// TwinCAT 3 PLC project EventsHistoricalSimple
// ProgramVersion: 3.1.4020.4
// CompilerDefines: VISU_USEWSTRING
// libraries:
//   Tc2_Standard, * (Beckhoff Automation GmbH)
//   Tc2_System, * (Beckhoff Automation GmbH)
//   Tc2_Utilities, * (Beckhoff Automation GmbH)
//   Tc3_Module, * (Beckhoff Automation GmbH)
//   VisuDialogs, * (System)
// project tree:
//   DUTsEventsHS/ ST_EventDefinition.TcDUT, ST_EventHistoricalSimple.TcDUT, ST_EventHistoricalSimplePersistent.TcDUT
//   / GlobalTextList.TcGTLO, PlcTask.TcTTO, Visualization Manager.TcVMO (not stored), VISU_TASK.TcTTO
//   GVLsEventsHS/ GVL_EHS.TcGVL, GVL_EHSP.TcGVL
//   POUsEventsHS/POUsEventsHS/Functions/ F_RESET_Event.TcPOU, F_SET_Event.TcPOU
//   POUsEventsHS/POUsEventsHS/ P_EventsHS.TcPOU, P_EventsDefinitionHS.TcPOU, P_EventsHandlingHS.TcPOU, P_EventsVisuHS.TcPOU
//   POUsEventsHS/ MAIN.TcPOU
//   VISUsEventsHS/ VISU_EventsHistoricalSimple.TcVIS
// real-time tasks:
//   TASK PlcTask: cycle T#10ms, priority 20, ADS port 350
//   TASK VISU_TASK: cycle T#100000us, priority 30, ADS port 351

CONFIGURATION EventsHistoricalSimple
    RESOURCE PLC ON TwinCAT3
        TASK PlcTask(INTERVAL := T#10ms, PRIORITY := 20);
        TASK VISU_TASK(INTERVAL := T#100000us, PRIORITY := 30);
        PROGRAM MAIN WITH PlcTask : MAIN;
        PROGRAM VisuElems_Visu_Prg WITH VISU_TASK : VisuElems.Visu_Prg;
    END_RESOURCE
END_CONFIGURATION

// ---- DUTsEventsHS/ST_EventDefinition.TcDUT
//==================================================================================================
//							Beckhoff Automation Poland
//									23.05.2017
//	Struktura zawierajaca definicje zdarzenia
// 	v1.0	|| TC v 3.1.4020.32		|| - pierwsza wersja
//==================================================================================================
TYPE ST_EventDefinition :
STRUCT
	dwClass									: DWORD;
	dwParam									: DWORD;
	wsMessage								: WSTRING(80);
	bActive									: BOOL;
END_STRUCT
END_TYPE

// ---- DUTsEventsHS/ST_EventHistoricalSimple.TcDUT
//==================================================================================================
//							Beckhoff Automation Poland
//									23.05.2017
//	Struktura zawierajaca zdarzenie - pelne informacje, np. do wizualizacji
// 	v1.0	|| TC v 3.1.4020.32		|| - pierwsza wersja
//==================================================================================================
TYPE ST_EventHistoricalSimple :
STRUCT
	dwID									: DWORD;
	dwParam									: DWORD;
	dwClass									: DWORD;
	dtDateBegin								: DT;
	dtDateEnd								: DT;
	wsMessage								: WSTRING(80);
	dwColor									: UDINT;
END_STRUCT
END_TYPE

// ---- DUTsEventsHS/ST_EventHistoricalSimplePersistent.TcDUT
//==================================================================================================
//							Beckhoff Automation Poland
//									23.05.2017
//	Struktura zawierajaca zane do przechowania zdarzenia w pamieci
// 	v1.0	|| TC v 3.1.4020.32		|| - pierwsza wersja
//==================================================================================================
TYPE ST_EventHistoricalSimplePersistent :
STRUCT
	dwID									: DWORD;
	dwParam									: DWORD;
	dwClass									: DWORD;
	dtDateBegin								: DT;
	dtDateEnd								: DT;
END_STRUCT
END_TYPE

// ---- GVLsEventsHS/GVL_EHS.TcGVL
//==================================================================================================
//							Beckhoff Automation Poland
//									23.05.2017
// 	v1.0	|| TC v 3.1.4020.32		|| - pierwsza wersja
//==================================================================================================
{attribute 'qualified_only'}
VAR_GLOBAL CONSTANT
	diEventsDefinition						: DINT 	:= 50;				// Rozmiar tablicy definicji zdarzen, powinna byc w zakresie 5..1000
	diNoOfEvents							: DINT 	:= 100;				// Rozmiar tablicy zdarzen historycznych, powinna byc w zakresie 5..1000
END_VAR
VAR_GLOBAL
	stActTime								: TIMESTRUCT;				// Aktualny czas sytemowy w formie struktury
	dtActTime								: DT;						// Aktualny czas sytemowy
	arrEventDefinition 						: ARRAY [1..GVL_EHS.diEventsDefinition] OF ST_EventDefinition;
	arrEventVisu							: ARRAY [1..GVL_EHS.diNoOfEvents] OF ST_EventHistoricalSimple;		// Pokazywane na wizualizacji - po filtracji
	dwLanguageId							: DWORD := 1033;			// Kod jezyka wyswietlania - Microsoft Locale ID Values
END_VAR

// ---- GVLsEventsHS/GVL_EHSP.TcGVL
//==================================================================================================
//							Beckhoff Automation Poland
//									23.05.2017
// 	v1.0	|| TC v 3.1.4020.32		|| - pierwsza wersja
//==================================================================================================
{attribute 'qualified_only'}
VAR_GLOBAL PERSISTENT
	arrEvent								: ARRAY [1..GVL_EHS.diNoOfEvents] OF ST_EventHistoricalSimplePersistent;
END_VAR

// ---- POUsEventsHS/MAIN.TcPOU
PROGRAM MAIN
VAR
	tonWritePersistent						: TON;
	fbPersistent 							: FB_WritePersistentData;
END_VAR

tonWritePersistent(IN:= NOT tonWritePersistent.Q, PT:= T#1M, Q=> , ET=> );		// Zapis persistentow
fbPersistent(PORT:= 851, START:= tonWritePersistent.Q);							// Zapis persistentow
P_EventsHS();

END_PROGRAM

// ---- POUsEventsHS/POUsEventsHS/P_EventsHS.TcPOU
//==================================================================================================
//							Beckhoff Automation Poland
//									23.05.2017
//	Program obslugujacy proste alarmy historyczne.
//	W opcjach wizualizacji trzeba wybrac use uniceode strings i use current visu variable
// 	v1.0	|| TC v 3.1.4020.32		|| - pierwsza wersja
//==================================================================================================
PROGRAM P_EventsHS
VAR
	fbLocalSystemTime						: FB_LocalSystemTime;
	bEventTableSizeError					: BOOL;					// Niewlasciwy rozmiar tablicy zdarzen - sprawdz GVL_EHS.diNoOfEvents
	bEventDefinitionSizeError				: BOOL;					// Niewlasciwy rozmiar tablicy zdarzen - sprawdz GVL_EHS.diEventsDefinition
END_VAR

fbLocalSystemTime(bEnable:= TRUE, systemTime=> GVL_EHS.stActTime);
GVL_EHS.dtActTime 							:= SYSTEMTIME_TO_DT(GVL_EHS.stActTime);

P_EventsDefinitionHS ();

bEventDefinitionSizeError 					:= GVL_EHS.diEventsDefinition < 5 OR GVL_EHS.diEventsDefinition > 1000;
bEventTableSizeError 						:= GVL_EHS.diNoOfEvents < 5 OR GVL_EHS.diNoOfEvents > 1000;

IF NOT bEventDefinitionSizeError AND NOT bEventTableSizeError THEN
	IF fbLocalSystemTime.bValid THEN
		P_EventsHandlingHS();
	END_IF
	// Visu i filtry
	P_EventsVisuHS();	
END_IF

END_PROGRAM

// ---- POUsEventsHS/POUsEventsHS/P_EventsDefinitionHS.TcPOU
//==================================================================================================
//							Beckhoff Automation Poland
//									23.05.2017
//	Program definiujacy zdarzenia - musi byc dostosowany do aplikacji
//	W pierwszym cyklu definiowane sa klasy
//	Zmiana jezyka na zdarzenie i w pierwszym cyklu
//	Wykrywanie aktywnosci zdarzenia i parametru - cykliczne
// 	v1.0	|| TC v 3.1.4020.32		|| - pierwsza wersja
//==================================================================================================
PROGRAM P_EventsDefinitionHS
VAR
	bFirstCycle 							: BOOL := TRUE;
	dwPreviousLanguageID					: DWORD;
END_VAR

// Class
IF bFirstCycle THEN
	ACT_ClassDefinition();
	bFirstCycle 							:= FALSE;
END_IF

// Language
ACT_Language();

// Active
ACT_Active();

ACTION ACT_1033_US:
GVL_EHS.arrEventDefinition[1].wsMessage	 	:= "Alarm Message 1";
GVL_EHS.arrEventDefinition[2].wsMessage 	:= "Alarm Message 2";
GVL_EHS.arrEventDefinition[31].wsMessage 	:= "Warning Message 1";
GVL_EHS.arrEventDefinition[32].wsMessage 	:= "Warning Message 2";
GVL_EHS.arrEventDefinition[41].wsMessage 	:= "Message 1";
GVL_EHS.arrEventDefinition[42].wsMessage 	:= "Message 2";
END_ACTION

ACTION ACT_1045_PL:
GVL_EHS.arrEventDefinition[1].wsMessage		:= "Tekst alarmu 1";
GVL_EHS.arrEventDefinition[2].wsMessage		:= "śćąęźżółń 2";
GVL_EHS.arrEventDefinition[31].wsMessage	:= "Tekst ostrzeżenia 1";
GVL_EHS.arrEventDefinition[32].wsMessage	:= "Tekst ostrzeżenia 2";
GVL_EHS.arrEventDefinition[41].wsMessage	:= "Komunikat 1";
GVL_EHS.arrEventDefinition[42].wsMessage	:= "Komunikat 2";
END_ACTION

ACTION ACT_Active:
GVL_EHS.arrEventDefinition[1].bActive; // S=;
GVL_EHS.arrEventDefinition[1].bActive;// R=;
GVL_EHS.arrEventDefinition[1].dwParam := 1;
GVL_EHS.arrEventDefinition[2].bActive;
GVL_EHS.arrEventDefinition[2].dwParam := 2;
GVL_EHS.arrEventDefinition[31].bActive;
GVL_EHS.arrEventDefinition[31].dwParam := 3;
GVL_EHS.arrEventDefinition[32].bActive;
GVL_EHS.arrEventDefinition[32].dwParam := 4;
GVL_EHS.arrEventDefinition[41].bActive;
GVL_EHS.arrEventDefinition[41].dwParam := 5;
GVL_EHS.arrEventDefinition[42].bActive;
GVL_EHS.arrEventDefinition[42].dwParam;
END_ACTION

ACTION ACT_ClassDefinition:
// Error - 0
GVL_EHS.arrEventDefinition[1].dwClass := 0;
GVL_EHS.arrEventDefinition[2].dwClass := 0;
GVL_EHS.arrEventDefinition[3].dwClass := 0;
GVL_EHS.arrEventDefinition[4].dwClass := 0;

// Warning - 1
GVL_EHS.arrEventDefinition[31].dwClass := 1;
GVL_EHS.arrEventDefinition[32].dwClass := 1;
GVL_EHS.arrEventDefinition[33].dwClass := 1;
GVL_EHS.arrEventDefinition[34].dwClass := 1;

// Message - 2
GVL_EHS.arrEventDefinition[41].dwClass := 2;
GVL_EHS.arrEventDefinition[42].dwClass := 2;
GVL_EHS.arrEventDefinition[43].dwClass := 2;
GVL_EHS.arrEventDefinition[44].dwClass := 2;
END_ACTION

ACTION ACT_Language:
// Wybor jezyka
IF dwPreviousLanguageID <> GVL_EHS.dwLanguageId THEN
	CASE GVL_EHS.dwLanguageId OF
		
		1033:	// United States
			ACT_1033_US();
			
		1045:	// Polish
			ACT_1045_PL();
	
	ELSE	// Default Polish
		
			ACT_1045_PL();
	END_CASE
END_IF

dwPreviousLanguageID := GVL_EHS.dwLanguageId;
END_ACTION

END_PROGRAM

// ---- POUsEventsHS/POUsEventsHS/P_EventsHandlingHS.TcPOU
//==================================================================================================
//							Beckhoff Automation Poland
//									23.05.2017
//	Program obslugujacy zdarzenia historyczne - edycji podlega tylko tRefreshTime i bRealTime
// 	v1.0	|| TC v 3.1.4020.32		|| - pierwsza wersja
//==================================================================================================
PROGRAM P_EventsHandlingHS
VAR
	bRealTime								: BOOL := TRUE;		// Odswiezanie ciagle - zmieniamy na FALSE tylko gdy jest duze obciazenie CPU
																// Zmiana na FLASE powoduje odfiltrowanie alarmow zgodnie z czasem tRefreshTime
	tonRefresh								: TON;				// Timer odswiezenia
	tRefreshTime							: TIME := T#1S;		// Czestotliwosc odswiezania - im dluzszy szac tym wieksze ryzyko niezauwazenia wystapienia alarmu
	bInitialized							: BOOL;				// Flaga inicjalizacji
	i										: DINT;				// Iterator petli
	// Tablice wykrycia poczatku/konca zdarzenia
	arrSet									: ARRAY [1..GVL_EHS.diEventsDefinition] OF R_TRIG;
	arrReset								: ARRAY [1..GVL_EHS.diEventsDefinition] OF F_TRIG;
END_VAR

// Inicjalizacja - po uruchomieniu znajdz niezakonczone alarmy i dodaj aktualny czas jako zakonczenie
IF NOT bInitialized THEN
	FOR i := 1 TO GVL_EHS.diEventsDefinition DO
		F_RESET_Event(dwID:= i, dtActTime:= GVL_EHS.dtActTime);
	END_FOR	
	bInitialized 							:= TRUE;
END_IF

// Timer odswiezania
tonRefresh(IN:= NOT tonRefresh.Q, PT:= tRefreshTime, Q=> , ET=> );

IF bRealTime OR tonRefresh.Q THEN
	FOR i := 1 TO GVL_EHS.diEventsDefinition DO
		// Wykrycie pojawienia sie zdarzenia - ustawienie flagi na 1 cykl i dodanie na poczatek listy
		arrSet[i](CLK:= GVL_EHS.arrEventDefinition[i].bActive);
		IF arrSet[i].Q THEN
			F_SET_Event(dwID:= i, stEventDefinition:= GVL_EHS.arrEventDefinition[i], dtActTime:= GVL_EHS.dtActTime);
		END_IF
		// Wykrycie zakonczenia zdarzenia - ustawienie flagi na 1 cykl i dodanie daty zakonczenia
		arrReset[i](CLK:= GVL_EHS.arrEventDefinition[i].bActive);
		IF arrReset[i].Q THEN
			F_RESET_Event(dwID:= i, dtActTime:= GVL_EHS.dtActTime);
		END_IF
	END_FOR	
END_IF

END_PROGRAM

// ---- POUsEventsHS/POUsEventsHS/Functions/F_RESET_Event.TcPOU
FUNCTION F_RESET_Event : BOOL
VAR_INPUT
	dwID									: DWORD;
	dtActTime								: DT;
END_VAR
VAR
	i										: DINT;
END_VAR

// Znajdz i wstaw date zakonczenia
FOR i := 1 TO GVL_EHS.diNoOfEvents DO
	IF 	GVL_EHSP.arrEvent[i].dwID = dwID THEN
		GVL_EHSP.arrEvent[i].dtDateEnd		:= dtActTime;
		EXIT;
	END_IF
END_FOR

END_FUNCTION

// ---- POUsEventsHS/POUsEventsHS/Functions/F_SET_Event.TcPOU
FUNCTION F_SET_Event : BOOL
VAR_INPUT
	dwID									: DWORD;
	stEventDefinition						: ST_EventDefinition;
	dtActTime								: DT;
END_VAR
VAR
	i										: DINT;
END_VAR

// Przesun elemety tablicy
FOR i := 0 TO GVL_EHS.diNoOfEvents-2 DO
	GVL_EHSP.arrEvent[GVL_EHS.diNoOfEvents-i] := GVL_EHSP.arrEvent[GVL_EHS.diNoOfEvents-i-1];
END_FOR
// Dodaj nowy
GVL_EHSP.arrEvent[1].dwID					:= dwID;
GVL_EHSP.arrEvent[1].dtDateBegin 			:= dtActTime;
GVL_EHSP.arrEvent[1].dtDateEnd	 			:= DT#1970-1-1-0:0:0;
GVL_EHSP.arrEvent[1].dwParam 				:= stEventDefinition.dwParam;
GVL_EHSP.arrEvent[1].dwClass 				:= stEventDefinition.dwClass;

END_FUNCTION

// ---- POUsEventsHS/POUsEventsHS/P_EventsVisuHS.TcPOU
//==================================================================================================
//							Beckhoff Automation Poland
//									23.05.2017
//	Program obslugujacy wizualizacje VISU_EventsHistoricalSimple
//	Mozliwe filtrowanie alamow. Czestotliwosc odswiezania wplywa tylko na wyswietlanie
// 	v1.0	|| TC v 3.1.4020.32		|| - pierwsza wersja
//==================================================================================================
PROGRAM P_EventsVisuHS
VAR
	i										: DINT;				// Iterator tablicy przechowywanej w pamieci
	j										: DINT;				// Iterator tablicy wyswietlanej
	bActiveWindow							: BOOL := TRUE;		// Flaga wysietlania okna - tylko wtedy odswiezamy tablice wyswietlana
	rtPageChange							: R_TRIG;			// Wykrycie przelaczenia strony
	tonRefresh								: TON;
	tRefreshTime							: TIME := T#50MS;	// Czestotliwosc odswiezania strony
	//========================= Filtry =========================
	bRemoveFromList							: BOOL; 			// Flaga pomocnicza dla filtrow - decyduje czy element ma byc dodany na wizualizacje
	// Flagi wykonywalnosci
	bFilterID								: BOOL;
	bFilterClass							: BOOL;
	bFilterBeginTimeFrom					: BOOL;
	bFilterBeginTimeTo						: BOOL;
	bFilterEndTimeFrom						: BOOL;
	bFilterEndTimeTo						: BOOL;
	bFilterActiveOnly						: BOOL;
	// Parametry
	dwFilterID								: DWORD;	
	dwFilterClass							: DWORD;
	dtFilterBeginTimeFrom					: DT;
	dtFilterBeginTimeTo						: DT;
	dtFilterEndTimeFrom						: DT;
	dtFilterEndTimeTo						: DT;

END_VAR

bActiveWindow := VisuElems.CURRENTVISU = 'VISU_EventsHistoricalSimple';						// Flaga wysietlania okna
rtPageChange(CLK:= bActiveWindow, Q=> );													// Wykrycie zmiany strony - jednorazowo inicjalizacja
tonRefresh(IN:= bActiveWindow AND NOT tonRefresh.Q, PT:= tRefreshTime, Q=> , ET=> );		// Timer odswiezania

IF  rtPageChange.Q OR tonRefresh.Q THEN
	// Czyszczenie tablicy
	MEMSET(ADR(GVL_EHS.arrEventVisu),0,SIZEOF(GVL_EHS.arrEventVisu));
	j := 1;
	// Filters
	FOR i := 1 TO GVL_EHS.diNoOfEvents DO
		bRemoveFromList 								:= FALSE;
		// Jesli jest element
		IF GVL_EHSP.arrEvent[i].dwID <> 0 THEN
			bRemoveFromList								:= bFilterID AND dwFilterID <> GVL_EHSP.arrEvent[i].dwID;
			bRemoveFromList								:= bRemoveFromList OR (bFilterClass AND dwFilterClass <> GVL_EHSP.arrEvent[i].dwClass);
			bRemoveFromList								:= bRemoveFromList OR (bFilterBeginTimeFrom AND GVL_EHSP.arrEvent[i].dtDateBegin <= dtFilterBeginTimeFrom);
			bRemoveFromList								:= bRemoveFromList OR (bFilterBeginTimeTo AND GVL_EHSP.arrEvent[i].dtDateBegin >= dtFilterBeginTimeTo);
			bRemoveFromList								:= bRemoveFromList OR (bFilterEndTimeFrom AND GVL_EHSP.arrEvent[i].dtDateEnd <= dtFilterEndTimeFrom);
			bRemoveFromList								:= bRemoveFromList OR (bFilterEndTimeTo AND GVL_EHSP.arrEvent[i].dtDateEnd >= dtFilterEndTimeTo);
			bRemoveFromList								:= bRemoveFromList OR (bFilterActiveOnly AND DT#1970-1-1-0:0:0 <> GVL_EHSP.arrEvent[i].dtDateEnd);
			// Analogicznie dodajemy inne filtry jesli jest taka potrzeba
			// Jesli element nie zostal usuniety przez filtr to dodajemy go do tablicy alarmow wyswietlanych
			IF NOT bRemoveFromList THEN
				GVL_EHS.arrEventVisu[j].dwID 			:= GVL_EHSP.arrEvent[i].dwID;
				GVL_EHS.arrEventVisu[j].dwClass 		:= GVL_EHSP.arrEvent[i].dwClass;
				GVL_EHS.arrEventVisu[j].wsMessage		:= GVL_EHS.arrEventDefinition[GVL_EHSP.arrEvent[i].dwID].wsMessage;
				GVL_EHS.arrEventVisu[j].dwParam 		:= GVL_EHSP.arrEvent[i].dwParam;
				GVL_EHS.arrEventVisu[j].dtDateBegin 	:= GVL_EHSP.arrEvent[i].dtDateBegin;
				GVL_EHS.arrEventVisu[j].dtDateEnd 		:= GVL_EHSP.arrEvent[i].dtDateEnd;
				IF GVL_EHS.arrEventVisu[j].dwClass=0 THEN
					GVL_EHS.arrEventVisu[j].dwColor:=16#FFDE6666;
				ELSIF GVL_EHS.arrEventVisu[j].dwClass=1 THEN
					GVL_EHS.arrEventVisu[j].dwColor:=16#FFF2F063;
				ELSIF GVL_EHS.arrEventVisu[j].dwClass=2 THEN
					GVL_EHS.arrEventVisu[j].dwColor:=16#FF6AD8EE;
				END_IF
				j := j + 1;
			END_IF
		END_IF
	END_FOR
END_IF

END_PROGRAM

// ---- GlobalTextList.TcGTLO
TEXTLIST GlobalTextList
  22 = '%s'
  6 = 'Active'
  20 = 'Active Only'
  7 = 'Alarm 1'
  8 = 'Alarm 2'
  2 = 'Class'
  3 = 'Date Begin'
  4 = 'Date End'
  14 = 'EN'
  0 = 'ID'
  5 = 'Message'
  11 = 'Message 1'
  12 = 'Message 2'
  1 = 'Param'
  13 = 'PL'
  21 = 'P_EventsVisu.bFilterActiveOnly'
  15 = 'T Begin From'
  16 = 'Time Begin From'
  17 = 'Time Begin To'
  18 = 'Time End From'
  19 = 'Time End To'
  9 = 'Warning 1'
  10 = 'Warning 2'
END_TEXTLIST

// ---- VISUsEventsHS/VISU_EventsHistoricalSimple.TcVIS
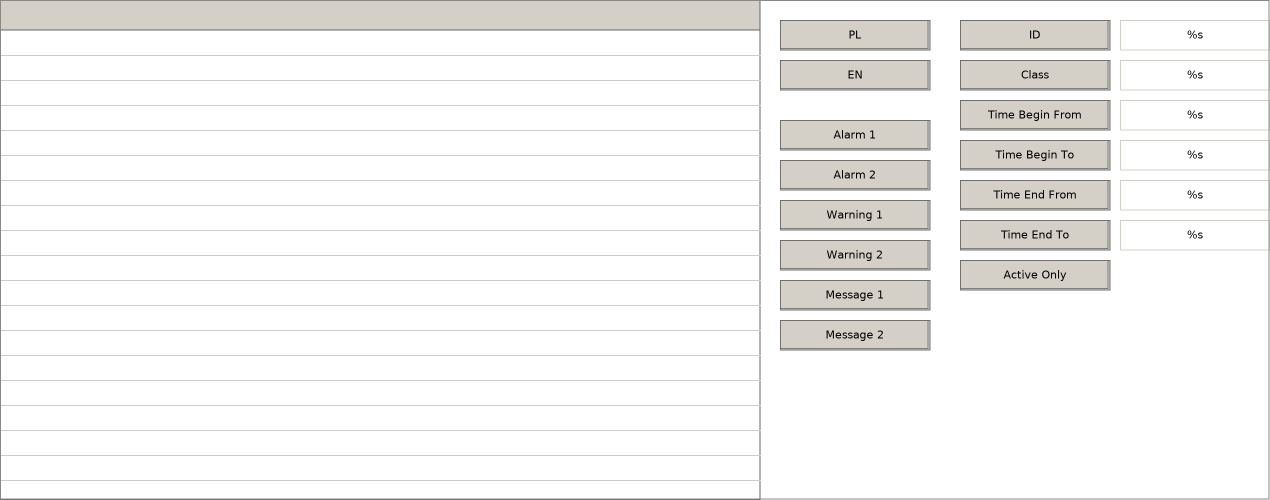
VISUALIZATION VISU_EventsHistoricalSimple  // 1270x500
    Group (780,120 150x230)
        Button (0,0 150x30), "Alarm 1", colour toggle: GVL_EHS.arrEventDefinition[1].bActive
            toggle GVL_EHS.arrEventDefinition[1].bActive
        Button (0,40 150x30), "Alarm 2", colour toggle: GVL_EHS.arrEventDefinition[2].bActive
            toggle GVL_EHS.arrEventDefinition[2].bActive
        Button (0,80 150x30), "Warning 1", colour toggle: GVL_EHS.arrEventDefinition[31].bActive
            toggle GVL_EHS.arrEventDefinition[31].bActive
        Button (0,120 150x30), "Warning 2", colour toggle: GVL_EHS.arrEventDefinition[32].bActive
            toggle GVL_EHS.arrEventDefinition[32].bActive
        Button (0,160 150x30), "Message 1", colour toggle: GVL_EHS.arrEventDefinition[41].bActive
            toggle GVL_EHS.arrEventDefinition[41].bActive
        Button (0,200 150x30), "Message 2", colour toggle: GVL_EHS.arrEventDefinition[42].bActive
            toggle GVL_EHS.arrEventDefinition[42].bActive
    Group (780,20 150x70)
        Button (0,0 150x30), "PL"
            OnMouseDown: execute { GVL_EHS.dwLanguageId := 1045; }
        Button (0,40 150x30), "EN"
            OnMouseDown: execute { GVL_EHS.dwLanguageId := 1033; }
    Table (0,0 760x500), data array: GVL_EHS.arrEventVisu
        p3854506369: GVL_EHS.arrEventVisu[INDEX].dwID
        p1892666644: GVL_EHS.arrEventVisu[INDEX].dwParam
        p338671338: GVL_EHS.arrEventVisu[INDEX].wsMessage
        p2170511999: GVL_EHS.arrEventVisu[INDEX].dtDateBegin
        p3723444502: GVL_EHS.arrEventVisu[INDEX].dtDateEnd
        p511219082: Class
        p2237128397: Date Begin
        p505689113: Date End
        p3312258591: GVL_EHS.arrEventVisu[INDEX].dwClass
        Columns.Column.[2].Template: GVL_EHS.arrEventVisu[INDEX].dwColor
    Group (960,20 310x270)
        Button (0,0 150x30), "ID", colour toggle: P_EventsVisuHS.bFilterID
            toggle P_EventsVisuHS.bFilterID
        Button (0,40 150x30), "Class", colour toggle: P_EventsVisuHS.bFilterClass
            toggle P_EventsVisuHS.bFilterClass
        Button (0,80 150x30), "Time Begin From", colour toggle: P_EventsVisuHS.bFilterBeginTimeFrom
            toggle P_EventsVisuHS.bFilterBeginTimeFrom
        Button (0,120 150x30), "Time Begin To", colour toggle: P_EventsVisuHS.bFilterBeginTimeTo
            toggle P_EventsVisuHS.bFilterBeginTimeTo
        Button (0,160 150x30), "Time End From", colour toggle: P_EventsVisuHS.bFilterEndTimeFrom
            toggle P_EventsVisuHS.bFilterEndTimeFrom
        Button (0,200 150x30), "Time End To", colour toggle: P_EventsVisuHS.bFilterEndTimeTo
            toggle P_EventsVisuHS.bFilterEndTimeTo
        Button (0,240 150x30), "Active Only", colour toggle: P_EventsVisuHS.bFilterActiveOnly
            toggle P_EventsVisuHS.bFilterActiveOnly
        Textfield (160,0 150x30), "%s", text variable: P_EventsVisuHS.dwFilterID
            OnMouseDown: write the text variable via VisuDialogs.Numpad
        Textfield (160,40 150x30), "%s", text variable: P_EventsVisuHS.dwFilterClass
            OnMouseDown: write the text variable via VisuDialogs.Numpad
        Textfield (160,80 150x30), "%s", text variable: P_EventsVisuHS.dtFilterBeginTimeFrom
            OnMouseDown: write the text variable via Edit
        Textfield (160,120 150x30), "%s", text variable: P_EventsVisuHS.dtFilterBeginTimeTo
            OnMouseDown: write the text variable via Edit
        Textfield (160,160 150x30), "%s", text variable: P_EventsVisuHS.dtFilterEndTimeFrom
            OnMouseDown: write the text variable via Edit
        Textfield (160,200 150x30), "%s", text variable: P_EventsVisuHS.dtFilterEndTimeTo
            OnMouseDown: write the text variable via Edit
END_VISUALIZATION
